TYPE ST_EventEntryTableListener EXTENDS ST_EventEntryTable:
STRUCT
	sJsonAttribute	: STRING(8000);
	ipArguments		: I_TcArguments;
END_STRUCT
END_TYPE

(* stored: Version 1.1.0.1, ProductVersion 3.1.4026.18
   DUT ST_EventEntryTableListener: Id {4e02f4c4-e85b-4a46-8864-8a81fbdaff13} *)
